(* PLC project Unnamed, Unknown Unnamed 1 *)
(* stored: creationDateTime 2023-06-04T11:47:30, modificationDateTime 2023-06-04T11:47:30 *)

CONFIGURATION Config0
  RESOURCE Res0 ON PLC
  END_RESOURCE
END_CONFIGURATION
